// TIA Portal V17 export
// export: Created 2023-08-28T22:41:32.6164324Z, ExportSetting WithDefaults, DisplayName Totally Integrated Automation Portal, DisplayVersion V17 Update 5, DisplayName TIA Portal Openness, DisplayVersion V17 Update 5, DisplayName TIA Portal Teamcenter Gateway, DisplayVersion V17 Update 5, DisplayName TIA Portal Version Control Interface, DisplayVersion V17, DisplayName Simotion SCOUT TIA, DisplayVersion 5.4.3.0, DisplayName TIA Portal Test Suite Advanced, DisplayVersion V17 Update 1, DisplayName SIMOCODE ES, DisplayVersion V17 Update 5, DisplayName SINAMICS Startdrive Advanced, DisplayVersion V17 SP1, DisplayName SINAMICS Startdrive G130, G150, S120, S150, SINAMICS MV, S210, DisplayVersion V17 SP1, DisplayName SINAMICS Startdrive G110M, G120, G120C, G120D, G120P, G115D, DisplayVersion V17 SP1, DisplayName SIRIUS Safety ES, DisplayVersion V17 Update 5, DisplayName STEP 7 Professional, DisplayVersion V17 Update 5, DisplayName STEP 7 CFC, DisplayVersion V17 Update 1, DisplayName STEP 7 Safety, DisplayVersion V17, DisplayName WinCC Advanced, DisplayVersion V17 Update 5, DisplayName SIMATIC Visualization Architect, DisplayVersion V17 Update 5
DATA_BLOCK "GATE_SE01-B1"   // DB2900
// stored: AutoNumber true, DBAccessibleFromOPCUA true, DBAccessibleFromWebserver true, InstanceOfName 02_Safety_Door, InstanceOfType FB
"02_Safety_Door "
BEGIN
END_DATA_BLOCK

DATA_BLOCK "GATE_SE01-B2"   // DB2901
// stored: AutoNumber true, DBAccessibleFromOPCUA true, DBAccessibleFromWebserver true, InstanceOfName 02_Safety_Door, InstanceOfType FB
"02_Safety_Door "
BEGIN
END_DATA_BLOCK

DATA_BLOCK "GATE_SE01-B3"   // DB2902
// stored: AutoNumber true, DBAccessibleFromOPCUA true, DBAccessibleFromWebserver true, InstanceOfName 02_Safety_Door, InstanceOfType FB
"02_Safety_Door "
BEGIN
END_DATA_BLOCK

DATA_BLOCK "GATE_SE01-B4"   // DB2903
// stored: AutoNumber true, DBAccessibleFromOPCUA true, DBAccessibleFromWebserver true, InstanceOfName 02_Safety_Door, InstanceOfType FB
"02_Safety_Door "
BEGIN
END_DATA_BLOCK

DATA_BLOCK "GATE_SE01-B5"   // DB2904
// stored: AutoNumber true, DBAccessibleFromOPCUA true, DBAccessibleFromWebserver true, InstanceOfName 02_Safety_Door, InstanceOfType FB
"02_Safety_Door "
BEGIN
END_DATA_BLOCK

DATA_BLOCK "GATE_SE01-B6"   // DB2905
// stored: AutoNumber true, DBAccessibleFromOPCUA true, DBAccessibleFromWebserver true, InstanceOfName 02_Safety_Door, InstanceOfType FB
"02_Safety_Door "
BEGIN
END_DATA_BLOCK

DATA_BLOCK "GATE_SE01-B7"   // DB2906
// stored: AutoNumber true, DBAccessibleFromOPCUA true, DBAccessibleFromWebserver true, InstanceOfName 02_Safety_Door, InstanceOfType FB
"02_Safety_Door "
BEGIN
END_DATA_BLOCK

DATA_BLOCK "GATE_SE01-B8"   // DB2907
// stored: AutoNumber true, DBAccessibleFromOPCUA true, DBAccessibleFromWebserver true, InstanceOfName 02_Safety_Door, InstanceOfType FB
"02_Safety_Door "
BEGIN
END_DATA_BLOCK

DATA_BLOCK "GATE_SE01-B9"   // DB2908
// stored: AutoNumber true, DBAccessibleFromOPCUA true, DBAccessibleFromWebserver true, InstanceOfName 02_Safety_Door, InstanceOfType FB
"02_Safety_Door "
BEGIN
END_DATA_BLOCK

DATA_BLOCK "GATE_SE01-B10"   // DB2909
// stored: AutoNumber true, DBAccessibleFromOPCUA true, DBAccessibleFromWebserver true, InstanceOfName 02_Safety_Door, InstanceOfType FB
"02_Safety_Door "
BEGIN
END_DATA_BLOCK

DATA_BLOCK "GATE_SE01-B11"   // DB2910
// stored: AutoNumber true, DBAccessibleFromOPCUA true, DBAccessibleFromWebserver true, InstanceOfName 02_Safety_Door, InstanceOfType FB
"02_Safety_Door "
BEGIN
END_DATA_BLOCK

DATA_BLOCK "GATE_SE01-B12"   // DB2911
// stored: AutoNumber true, DBAccessibleFromOPCUA true, DBAccessibleFromWebserver true, InstanceOfName 02_Safety_Door, InstanceOfType FB
"02_Safety_Door "
BEGIN
END_DATA_BLOCK

DATA_BLOCK "GATE_SC00+UC114.VS019"   // DB2912
// stored: AutoNumber true, DBAccessibleFromOPCUA true, DBAccessibleFromWebserver true, InstanceOfName 02_Safety_Door, InstanceOfType FB
"02_Safety_Door "
BEGIN
END_DATA_BLOCK

DATA_BLOCK "GATE_SC00+UC124.VS019"   // DB2913
// stored: AutoNumber true, DBAccessibleFromOPCUA true, DBAccessibleFromWebserver true, InstanceOfName 02_Safety_Door, InstanceOfType FB
"02_Safety_Door "
BEGIN
END_DATA_BLOCK

DATA_BLOCK "GATE_SC00+UC134.VS019"   // DB2914
// stored: AutoNumber true, DBAccessibleFromOPCUA true, DBAccessibleFromWebserver true, InstanceOfName 02_Safety_Door, InstanceOfType FB
"02_Safety_Door "
BEGIN
END_DATA_BLOCK

DATA_BLOCK "GATE_SC00+UC144.VS019"   // DB2915
// stored: AutoNumber true, DBAccessibleFromOPCUA true, DBAccessibleFromWebserver true, InstanceOfName 02_Safety_Door, InstanceOfType FB
"02_Safety_Door "
BEGIN
END_DATA_BLOCK

DATA_BLOCK "GATE_SC00+UC154.VS019"   // DB2916
// stored: AutoNumber true, DBAccessibleFromOPCUA true, DBAccessibleFromWebserver true, InstanceOfName 02_Safety_Door, InstanceOfType FB
"02_Safety_Door "
BEGIN
END_DATA_BLOCK

DATA_BLOCK "GATE_SC00+UC164.VS019"   // DB2917
// stored: AutoNumber true, DBAccessibleFromOPCUA true, DBAccessibleFromWebserver true, InstanceOfName 02_Safety_Door, InstanceOfType FB
"02_Safety_Door "
BEGIN
END_DATA_BLOCK

DATA_BLOCK "GATE_SC00+UC175.VS019"   // DB2918
// stored: AutoNumber true, DBAccessibleFromOPCUA true, DBAccessibleFromWebserver true, InstanceOfName 02_Safety_Door, InstanceOfType FB
"02_Safety_Door "
BEGIN
END_DATA_BLOCK

DATA_BLOCK "GATE_SC00+UC214.VS019"   // DB2919
// stored: AutoNumber true, DBAccessibleFromOPCUA true, DBAccessibleFromWebserver true, InstanceOfName 02_Safety_Door, InstanceOfType FB
"02_Safety_Door "
BEGIN
END_DATA_BLOCK

DATA_BLOCK "GATE_SC00+UC224.VS019"   // DB2920
// stored: AutoNumber true, DBAccessibleFromOPCUA true, DBAccessibleFromWebserver true, InstanceOfName 02_Safety_Door, InstanceOfType FB
"02_Safety_Door "
BEGIN
END_DATA_BLOCK

DATA_BLOCK "GATE_SC00+UC234.VS019"   // DB2921
// stored: AutoNumber true, DBAccessibleFromOPCUA true, DBAccessibleFromWebserver true, InstanceOfName 02_Safety_Door, InstanceOfType FB
"02_Safety_Door "
BEGIN
END_DATA_BLOCK

DATA_BLOCK "GATE_SC00+UC244.VS019"   // DB2922
// stored: AutoNumber true, DBAccessibleFromOPCUA true, DBAccessibleFromWebserver true, InstanceOfName 02_Safety_Door, InstanceOfType FB
"02_Safety_Door "
BEGIN
END_DATA_BLOCK

DATA_BLOCK "GATE_SC00+UC254.VS019"   // DB2923
// stored: AutoNumber true, DBAccessibleFromOPCUA true, DBAccessibleFromWebserver true, InstanceOfName 02_Safety_Door, InstanceOfType FB
"02_Safety_Door "
BEGIN
END_DATA_BLOCK

DATA_BLOCK "GATE_SC00+UC264.VS019"   // DB2924
// stored: AutoNumber true, DBAccessibleFromOPCUA true, DBAccessibleFromWebserver true, InstanceOfName 02_Safety_Door, InstanceOfType FB
"02_Safety_Door "
BEGIN
END_DATA_BLOCK

DATA_BLOCK "GATE_SC00+UC273.VS024"   // DB2925
// stored: AutoNumber true, DBAccessibleFromOPCUA true, DBAccessibleFromWebserver true, InstanceOfName 02_Safety_Door, InstanceOfType FB
"02_Safety_Door "
BEGIN
END_DATA_BLOCK

DATA_BLOCK "GATE_SF00+UF511.VS015"   // DB2926
// stored: AutoNumber true, DBAccessibleFromOPCUA true, DBAccessibleFromWebserver true, InstanceOfName 02_Safety_Door, InstanceOfType FB
"02_Safety_Door "
BEGIN
END_DATA_BLOCK
